(* IEC 61131-3 sources: CodesysTest/export/UN00 - Sharp Bagger/EM01 - Bagger Head/CM06 - Vacuum Bag Open/FB_PneumaticVacuumCups.pou, 1 file *)

(* ---- FB_PneumaticVacuumCups.pou.st ---- *)
(*#-#-#-#-#-#-#-#-#-#---Declaration---#-#-#-#-#-#-#-#-#-#-#-#-#*)

FUNCTION_BLOCK FB_PneumaticVacuumCups EXTENDS FB_BaseComponent IMPLEMENTS IVacuumBagOpen
VAR_INPUT

END_VAR
VAR_OUTPUT

END_VAR
VAR
	_vacuumOn : BOOL;
END_VAR
VAR_IN_OUT
	vacGenerator : FB_VacuumGenerator;
END_VAR(*#-#-#-#-#-#-#-#-#-#---Implementation---#-#-#-#-#-#-#-#-#-#-#-#-#*)

SUPER^();
